PROGRAM MAIN
VAR
	



isim:ARRAY[0..70] OF STRING;
kullanici: ARRAY[0..70] OF STRING;
sifreler: ARRAY[0..70] OF STRING;
soyisim:ARRAY[0..70] OF STRING;
gunler:ARRAY[1..7] OF BOOL;

ad:STRING;
soyad:STRING;
kuladi:STRING;
sifre:STRING;

kaydet:BOOL;







uyelik:BOOL;
uyelik1:BOOL;
sayici:INT;



giris:BOOL;




yenikul:STRING;
yenisifre:STRING;





msgtype:MESSAGEBOXDIALOG_TYPES;
msgtitle:STRING;
msgtxt:STRING;



i: INT;
j:INT;
	
	cikis: BOOL;
	

	

	saydir: R_TRIG;
	cikis2: BOOL;
	sayici1: INT;
	kaydet2: BOOL;
	sayici2: INT;
	g: INT;
	sayici3: INT;
	h: INT;
	n: INT;
	giris1: BOOL;
	
	mesai_saat_saydirici: R_TRIG;
	
END_VAR



msgtitle:='İşlem Durumu ';
msgtxt:='Kayıt İşlemi Başarılı..';


GVL_personel_kayit.messagetext:='Kayıt İşlemi Başarılı.. Mesai Ücreti Hesaplamak Mesai Günü Seç  Butonuna Basınız.';
GVL_personel_kayit.messagetitle:='Kayıt İşlemi Durumu';






Giris_Panel();
uyelik_panel();
Kayit_Sayfa();
mesai_gun();
mesai_saat();
Hesap_Panel();

ACTION Giris_Panel:

giris1:=FALSE;

IF GVL_personel_kayit.perMesaiGun THEN
	GVL_personel_kayit.dogru:=TRUE;
	
END_IF


IF giris=TRUE THEN
	
FOR n:=1 TO 70 BY 1 DO
	
  IF kullanici[n]=kuladi AND sifreler[n]=sifre AND NOT GVL_personel_kayit.dogru THEN
	  
 
	  VisuElems.CurrentVisu := 'Kayit_Sayfa';
	  
	  
	  
	 
  END_IF

  	
END_FOR

	
END_IF
END_ACTION

ACTION Hesap_Panel:

GVL_mesai_saat.mesaiucret:=50;
GVL_hesapSayfa.saydir1(IN:=GVL_hesapSayfa.start , PT:=T#10S , Q=>GVL_hesapSayfa.cikis , ET=>GVL_hesapSayfa.gecensure );

GVL_hesapSayfa.start:=TRUE;



IF GVL_hesapSayfa.cikis=TRUE THEN
	
 IF 
	 GVL_mesai_gun.pazartesi=TRUE  OR  GVL_mesai_gun.sali=TRUE OR  GVL_mesai_gun.carsamba=TRUE OR  GVL_mesai_gun.persembe=TRUE OR  GVL_mesai_gun.cuma=TRUE THEN
	
	
(*   IF GVL_mesai_saat.baslangicsaat < GVL_mesai_saat.bitissaat  THEN
    	GVL_hesapSayfa.hesaplama:= GVL_mesai_saat.bitissaat-GVL_mesai_saat.baslangicsaat;
		ELSE			
		GVL_hesapSayfa.hesaplama:=GVL_mesai_saat.baslangicsaat-GVL_mesai_saat.bitisdakika;
		
 
 
END_IF
 *)
	
	
	
 
 END_IF
 
 
 
 

 
(*  IF GVL_mesai_gun.cumartesi OR GVL_mesai_gun.pazar THEN
	 	
   	 
 GVL_hesapSayfa.hesaplama:= GVL_mesai_saat.bitisdakika-GVL_mesai_saat.baslangicdakika;
 
 
 END_IF
 *)
 
 
 



	
END_IF
END_ACTION

ACTION Kayit_sayfa:


GVL_personel_kayit.saydirici(CLK:=GVL_personel_kayit.kaydet , Q=>GVL_personel_kayit.cikis3 );

IF GVL_personel_kayit.kaydet THEN
	GVL_personel_kayit.invisibleKayit:=TRUE;
END_IF

IF VisuElems.CurrentVisu='mesaigunleri_sayfa'THEN
	GVL_personel_kayit.invisibleKayit:=FALSE;
END_IF


IF GVL_personel_kayit.kaydet=TRUE THEN
	
IF GVL_personel_kayit.cikis3=TRUE THEN
 
GVL_personel_kayit.sayac:=GVL_personel_kayit.sayac +1;

END_IF



FOR GVL_personel_kayit.i:=1 TO 70 BY 1 DO
	
IF GVL_personel_kayit.personelisim[GVL_personel_kayit.i] ='' THEN
	GVL_personel_kayit.personelisim[GVL_personel_kayit.i]:=GVL_personel_kayit.perisim;
		
ELSE
	GVL_personel_kayit.personelisim[GVL_personel_kayit.sayac]:=GVL_personel_kayit.perisim;
	
END_IF

EXIT;
END_FOR






IF GVL_personel_kayit.cikis3=TRUE THEN
	
	GVL_personel_kayit.sayac1:=GVL_personel_kayit.sayac1+1;		
END_IF

FOR GVL_personel_kayit.j:=1 TO 70 BY  1 DO
	
IF GVL_personel_kayit.personelsoyisim[GVL_personel_kayit.j]='' THEN
	GVL_personel_kayit.personelsoyisim[GVL_personel_kayit.j]:=GVL_personel_kayit.perSoyisim;
	ELSE
		GVL_personel_kayit.personelsoyisim[GVL_personel_kayit.sayac]:=GVL_personel_kayit.perSoyisim;
	
END_IF

EXIT;

END_FOR



IF GVL_personel_kayit.cikis3=TRUE THEN
	GVL_personel_kayit.sayac2:=GVL_personel_kayit.sayac2 +1;
	
END_IF

FOR GVL_personel_kayit.g:=1 TO 70 BY 1 DO
	
	IF GVL_personel_kayit.personelid[GVL_personel_kayit.g]='' THEN
		GVL_personel_kayit.personelid[GVL_personel_kayit.g]:=GVL_personel_kayit.perid;
		ELSE
		GVL_personel_kayit.personelid[GVL_personel_kayit.sayac2]:=GVL_personel_kayit.perid;	
		
	END_IF
	EXIT;
	
END_FOR



















END_IF




IF GVL_personel_kayit.temizle=TRUE THEN
	GVL_personel_kayit.perisim:='';
	GVL_personel_kayit.perSoyisim:='';
	GVL_personel_kayit.perid:='';
	
	
	
	


END_IF
END_ACTION

ACTION mesai_gun:





IF GVL_mesai_gun.pazartesi=TRUE THEN
	
	
GVL_mesai_gun.sali:=FALSE;
GVL_mesai_gun.carsamba:=FALSE;
GVL_mesai_gun.persembe:=FALSE;
GVL_mesai_gun.cuma:=FALSE;
GVL_mesai_gun.cumartesi:=FALSE;
GVL_mesai_gun.pazar:=FALSE;


END_IF






IF GVL_mesai_gun.sali=TRUE THEN
	
	
GVL_mesai_gun.pazartesi:=FALSE;
GVL_mesai_gun.carsamba:=FALSE;
GVL_mesai_gun.persembe:=FALSE;
GVL_mesai_gun.cuma:=FALSE;
GVL_mesai_gun.cumartesi:=FALSE;
GVL_mesai_gun.pazar:=FALSE;


END_IF





IF GVL_mesai_gun.carsamba=TRUE THEN
	
	
GVL_mesai_gun.pazartesi:=FALSE;
GVL_mesai_gun.sali:=FALSE;
GVL_mesai_gun.persembe:=FALSE;
GVL_mesai_gun.cuma:=FALSE;
GVL_mesai_gun.cumartesi:=FALSE;
GVL_mesai_gun.pazar:=FALSE;


END_IF




IF GVL_mesai_gun.persembe=TRUE THEN
	
	
GVL_mesai_gun.pazartesi:=FALSE;
GVL_mesai_gun.sali:=FALSE;
GVL_mesai_gun.carsamba:=FALSE;
GVL_mesai_gun.cuma:=FALSE;
GVL_mesai_gun.cumartesi:=FALSE;
GVL_mesai_gun.pazar:=FALSE;


END_IF





IF GVL_mesai_gun.cuma=TRUE THEN
	
	
GVL_mesai_gun.pazartesi:=FALSE;
GVL_mesai_gun.sali:=FALSE;
GVL_mesai_gun.carsamba:=FALSE;
GVL_mesai_gun.persembe:=FALSE;
GVL_mesai_gun.cumartesi:=FALSE;
GVL_mesai_gun.pazar:=FALSE;


END_IF






IF GVL_mesai_gun.cumartesi=TRUE THEN
	
	
GVL_mesai_gun.pazartesi:=FALSE;
GVL_mesai_gun.sali:=FALSE;
GVL_mesai_gun.carsamba:=FALSE;
GVL_mesai_gun.persembe:=FALSE;
GVL_mesai_gun.cuma:=FALSE;
GVL_mesai_gun.pazar:=FALSE;


END_IF
IF GVL_mesai_gun.pazar=TRUE THEN
	
	
GVL_mesai_gun.pazartesi:=FALSE;
GVL_mesai_gun.sali:=FALSE;
GVL_mesai_gun.carsamba:=FALSE;
GVL_mesai_gun.persembe:=FALSE;
GVL_mesai_gun.cumartesi:=FALSE;
GVL_mesai_gun.cuma:=FALSE;


END_IF
END_ACTION

ACTION mesai_saat:



GVL_mesai_saat.a:=FALSE;
GVL_mesai_saat.b:=FALSE;
GVL_mesai_saat.c:=FALSE;




 // Başlangıç Dakikası
IF GVL_mesai_saat.kaydet=TRUE THEN
	

	 
  
	IF GVL_mesai_saat.x1bslangicSaat>GVL_mesai_saat.x1bitisSaat THEN
	
	GVL_mesai_saat.x1_mesaiSaat:=GVL_mesai_saat.x1bslangicSaat-GVL_mesai_saat.x1bitisSaat;
	GVL_mesai_saat.a:=TRUE;
	ELSE
		
	GVL_mesai_saat.x1_mesaiSaat:=GVL_mesai_saat.x1bitisSaat-GVL_mesai_saat.x1bslangicSaat;
	GVL_mesai_saat.b:=TRUE;
	
	END_IF
 



	IF GVL_mesai_saat.x1_5bslangicSaat>GVL_mesai_saat.x1_5bitisSaat THEN
	
	GVL_mesai_saat.x1_5mesaiSaat:=(GVL_mesai_saat.x1_5bslangicSaat-GVL_mesai_saat.x1_5bitisSaat)*1.5;
	GVL_mesai_saat.c:=TRUE;
	
	ELSE
		
	
	GVL_mesai_saat.x1_5mesaiSaat := (GVL_mesai_saat.x1_5bitisSaat-GVL_mesai_saat.x1_5bslangicSaat)*1.5;
	GVL_mesai_saat.d:=TRUE;
	
	END_IF


	
     
	 




	IF GVL_mesai_saat.x3bslangicSaat>GVL_mesai_saat.x3bitisSaat THEN
	
	GVL_mesai_saat.x_3mesaiSaat:=(GVL_mesai_saat.x3bslangicSaat-GVL_mesai_saat.x3bitisSaat)*3;
	GVL_mesai_saat.e:=TRUE;
	ELSE
		
	GVL_mesai_saat.x_3mesaiSaat:=(GVL_mesai_saat.x3bitisSaat-GVL_mesai_saat.x3bslangicSaat)*3;
	GVL_mesai_saat.f:=TRUE;
	
	END_IF
	
	
	
	
	
	IF GVL_mesai_saat.a=TRUE  OR GVL_mesai_saat.b=TRUE  THEN
		GVL_mesai_saat.mesaiSaaat:=GVL_mesai_saat.x1_mesaiSaat;
		
	END_IF
	
	
	
	(* IF GVL_mesai_saat.c=TRUE  OR GVL_mesai_saat.d=TRUE  THEN
		
		GVL_mesai_saat.mesaiSaaat:=GVL_mesai_saat.x1_5mesaiSaat;
	END_IF
	
	IF GVL_mesai_saat.e=TRUE OR GVL_mesai_saat.f=TRUE THEN
		
		GVL_mesai_saat.mesaiSaaat:=GVL_mesai_saat.x_3mesaiSaat;
	END_IF *)
	
	GVL_mesai_saat.tum_mesai:=(GVL_mesai_saat.x1_mesaiSaat+GVL_mesai_saat.x1_5mesaiSaat+GVL_mesai_saat.x_3mesaiSaat);
 
	
	
	


END_IF
END_ACTION

ACTION Mesai_Ucret_Panel:



GVL_Mesai_Ucret.online:=TRUE;
END_ACTION

ACTION uyelik_panel:


saydir(CLK:=kaydet , Q=>cikis );
		
		

IF kaydet=TRUE THEN




IF cikis=TRUE THEN
	sayici:=sayici+1;
END_IF

	FOR i:=1 TO 70 BY 1 DO
	
		IF isim[i]='' THEN			
			isim[i]:=ad;
		ELSE
			isim[sayici]:=ad;
		END_IF
		
		EXIT;
		
	END_FOR



IF cikis=TRUE THEN
	sayici1:=sayici1+1;
END_IF



FOR j:=1 TO 70 BY 1 DO
	
  IF soyisim[j]='' THEN
	  soyisim[j]:=soyad;
   ELSE
	soyisim[sayici1]:=soyad;
  END_IF


EXIT;
END_FOR










IF cikis=TRUE THEN
	sayici2:=sayici2+1;
	END_IF



FOR g:=1 TO 70 BY 1 DO
	
  IF kullanici[g]='' THEN
	  kullanici[g]:=yenikul;
	  ELSE
		  kullanici[sayici2]:=yenikul;
  END_IF


EXIT;
END_FOR







IF cikis=TRUE THEN
	sayici3:=sayici3+1;
	END_IF



FOR h:=1 TO 70 BY 1 DO
	
  IF sifreler[h]='' THEN
	  sifreler[h]:=yenisifre;
	  ELSE
		  sifreler[sayici3]:=yenisifre;
  END_IF


EXIT;
END_FOR


























	

END_IF
END_ACTION

END_PROGRAM

(* stored: Version 1.1.0.1, ProductVersion 3.1.4024.12
   POU MAIN: Id {3939e62a-e95d-4b0e-8449-9e559d02c21b}, SpecialFunc None
   Action Giris_Panel: Id {b3dd225c-0cda-409c-88cf-e22b0339c929}
   Action Hesap_Panel: Id {e55e8e4c-b275-4488-a58f-320fa1569264}
   Action Kayit_sayfa: Id {4a3b87f7-ac59-4d93-8283-157cde9e917a}
   Action mesai_gun: Id {040defbb-62af-418d-b4ab-2dc951da809f}
   Action mesai_saat: Id {26c797ba-1eab-4dd7-8c5d-215e979778b4}
   Action Mesai_Ucret_Panel: Id {90767ff7-2000-4461-b0f5-8590c5c2ea1a}
   Action uyelik_panel: Id {37d547a8-df21-4636-91aa-1f574a517ccc} *)
